Yaskawa INFORM job: cone_nozzle_cone_program.JBI

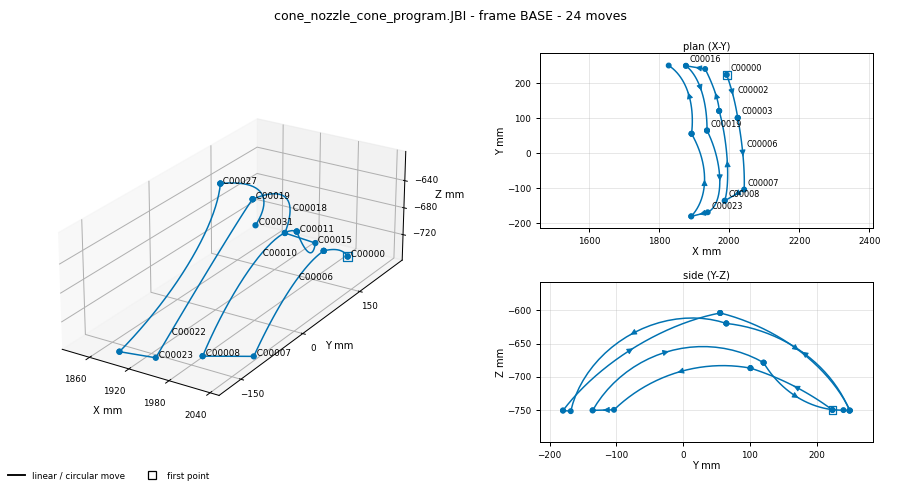
[picture p0: tool path of cone_nozzle_cone_program.JBI in frame BASE, 24 of 42 moves have a stored position in this frame; points joined in program order, loops and branches not executed]
/JOB
//NAME cone_nozzle_cone_program
//POS
///NPOS 32,0,32,0,0,0
///TOOL 0
///POSTYPE BASE
///RECTAN
///RCONF 0,0,0,0,0,0,0,0,0,0,0,0,0,0,0,0,0,0,0,0,0,0,0,0
C00000=1992.742256,223.779102,-749.556924,180.000000,-60.000000,-84.112206
C00001=1992.742256,223.779102,-749.556924,180.000000,-60.000000,-84.112206
C00002=2012.138122,161.510936,-711.422780,-175.000000,-38.482317,-91.264913
C00003=2024.514336,100.955294,-686.912521,164.399974,5.020513,-5.000000
C00004=2024.514336,100.955294,-686.912521,164.399974,5.020513,-5.000000
C00005=2024.514336,100.955294,-686.912521,164.399974,5.020513,-5.000000
C00006=2038.282018,6.567568,-689.267946,-161.138865,9.490423,5.000000
C00007=2042.865797,-103.517670,-749.344203,180.000000,-60.000000,101.560668
C00008=1987.501630,-135.481158,-750.149219,-180.000000,-60.000000,98.160892
C00009=1987.501630,-135.481158,-750.149219,-180.000000,-60.000000,98.160892
C00010=1993.889717,-10.132471,-658.827058,-160.727791,9.503494,5.000000
C00011=1971.663807,120.615731,-678.730431,155.831346,5.000000,-5.000000
C00012=1971.663807,120.615731,-678.730431,155.831346,5.000000,-5.000000
C00013=1971.663807,120.615731,-678.730431,155.831346,5.000000,-5.000000
C00014=1951.715836,196.075809,-742.508023,175.000000,-57.570601,-86.419290
C00015=1931.729073,240.213281,-749.792251,180.000000,-60.000000,-81.278669
C00016=1876.855673,249.294694,-750.558145,180.000000,-60.000000,-80.372601
C00017=1876.855673,249.294694,-750.558145,180.000000,-60.000000,-80.372601
C00018=1903.243575,218.333753,-699.434290,175.000000,-53.644239,-87.199948
C00019=1936.994429,64.747809,-619.928606,174.072397,6.814871,-5.000000
C00020=1936.994429,64.747809,-619.928606,174.072397,6.814871,-5.000000
C00021=1936.994429,64.747809,-619.928606,174.072397,6.814871,-5.000000
C00022=1952.347056,-158.016699,-721.088704,180.000000,-60.000000,101.388416
C00023=1939.012469,-168.286771,-751.377980,180.000000,-60.000000,97.328550
C00024=1891.924243,-179.956699,-750.416177,180.000000,-60.000000,96.809620
C00025=1891.924243,-179.956699,-750.416177,180.000000,-60.000000,96.809620
C00026=1908.416955,-158.160334,-724.657491,-175.000000,-63.894990,102.273265
C00027=1892.910649,55.576853,-604.248128,174.942063,6.961906,-5.000000
C00028=1892.910649,55.576853,-604.248128,174.942063,6.961906,-5.000000
C00029=1892.910649,55.576853,-604.248128,174.942063,6.961906,-5.000000
C00030=1851.821991,229.105814,-715.780159,175.000000,-61.145456,-85.766350
C00031=1827.720299,250.086305,-750.323790,180.000000,-60.000000,-79.820392
///POSTYPE PULSE
///PULSE
EX00000=0
EX00001=92160
EX00002=184320
EX00003=276480
///POSTYPE PULSE
///PULSE
EC00000=92160
EC00001=92160
EC00002=92160
EC00003=92160
EC00004=92160
EC00005=92160
EC00006=92160
EC00007=92160
EC00008=92160
EC00009=92160
EC00010=92160
EC00011=92160
EC00012=92160
EC00013=92160
EC00014=92160
EC00015=92160
EC00016=92160
EC00017=92160
EC00018=92160
EC00019=92160
EC00020=92160
EC00021=92160
EC00022=92160
EC00023=92160
EC00024=92160
EC00025=92160
EC00026=92160
EC00027=92160
EC00028=92160
EC00029=92160
EC00030=92160
EC00031=92160
//INST
///DATE 2023/08/07 14:10
///ATTR SC,RW,RJ
////FRAME BASE
///GROUP1 RB1,ST1
NOP
MOVJ P009 EX000 VJ=15.00
MOVJ P009 VJ=15.00
MOVJ P009 VJ=15.00
MOVL P009 EX00000 V=150.0
MOVJ C00000 EC00000 VJ=15.0
CALL JOB:SPYON
MOVC C00001 EC00001 V=150.0
MOVC C00002 EC00002 V=150.0
MOVC C00003 EC00003 V=150.0
MOVL C00004 EC00004 V=150.0
MOVC C00005 EC00005 V=150.0
MOVC C00006 EC00006 V=150.0
MOVC C00007 EC00007 V=150.0
MOVL C00008 EC00008 V=150.0
MOVC C00009 EC00009 V=150.0
MOVC C00010 EC00010 V=150.0
MOVC C00011 EC00011 V=150.0
MOVL C00012 EC00012 V=150.0
MOVC C00013 EC00013 V=150.0
MOVC C00014 EC00014 V=150.0
MOVC C00015 EC00015 V=150.0
MOVL C00016 EC00016 V=150.0
MOVC C00017 EC00017 V=150.0
MOVC C00018 EC00018 V=150.0
MOVC C00019 EC00019 V=150.0
MOVL C00020 EC00020 V=150.0
MOVC C00021 EC00021 V=150.0
MOVC C00022 EC00022 V=150.0
MOVC C00023 EC00023 V=150.0
MOVL C00024 EC00024 V=150.0
MOVC C00025 EC00025 V=150.0
MOVC C00026 EC00026 V=150.0
MOVC C00027 EC00027 V=150.0
MOVL C00028 EC00028 V=150.0
MOVC C00029 EC00029 V=150.0
MOVC C00030 EC00030 V=150.0
MOVC C00031 EC00031 V=150.0
CALL JOB:SPYOF
MOVJ P009 VJ=15.00
MOVL P009 EX00001 V=150.0
MOVJ P009 VJ=15.00
MOVL P009 EX00002 V=150.0
MOVJ P009 VJ=15.00
MOVL P009 EX00003 V=150.0
END
